TYPE M2MoveStepsProcedureStatuses :
STRUCT
	///Is the M2MoveStepsProcedure in a busy state?
	busyStatus: BusyStatus;
	///Is the M2MoveStepsProcedure in a healthy state?
	healthStatus: HealthStatus;
END_STRUCT
END_TYPE

(* stored: Version 1.1.0.1, ProductVersion 3.1.4019.2
   DUT M2MoveStepsProcedureStatuses: Id {2e31df31-19ce-43ea-90d2-5ed031b9f00a} *)
